# EPICS autosave request: opticsApp/Db/xia_slit_settings.req
# FILE...  xia_slit_settings.req
# USAGE... xia_slit.db fields to autosave

$(P)$(HSC)hID
$(P)$(HSC)vID
$(P)$(HSC)hOrient
$(P)$(HSC)vOrient
$(P)$(HSC)debug
$(P)$(HSC)l_tweakVal.VAL
$(P)$(HSC)r_tweakVal.VAL
$(P)$(HSC)width_tweakVal.VAL
$(P)$(HSC)height_tweakVal.VAL
$(P)$(HSC)t_tweakVal.VAL
$(P)$(HSC)b_tweakVal.VAL
$(P)$(HSC)h0_tweakVal.VAL
$(P)$(HSC)v0_tweakVal.VAL
